// SIMATIC S7-200 SMART project (STEP 7-Micro/WIN SMART), CPU SR40

SYMBOL_TABLE 表格 1
流速               VD116
管道内静压            VD112
管道内温度            VD108
管道内部压差值          VD104
粉尘浓度值            VD100
END_SYMBOL_TABLE

SYMBOL_TABLE 系统符号
Always_On        SM0.0    // 始终接通
END_SYMBOL_TABLE

ORGANIZATION_BLOCK MAIN:OB1
TITLE=程序注释
BEGIN
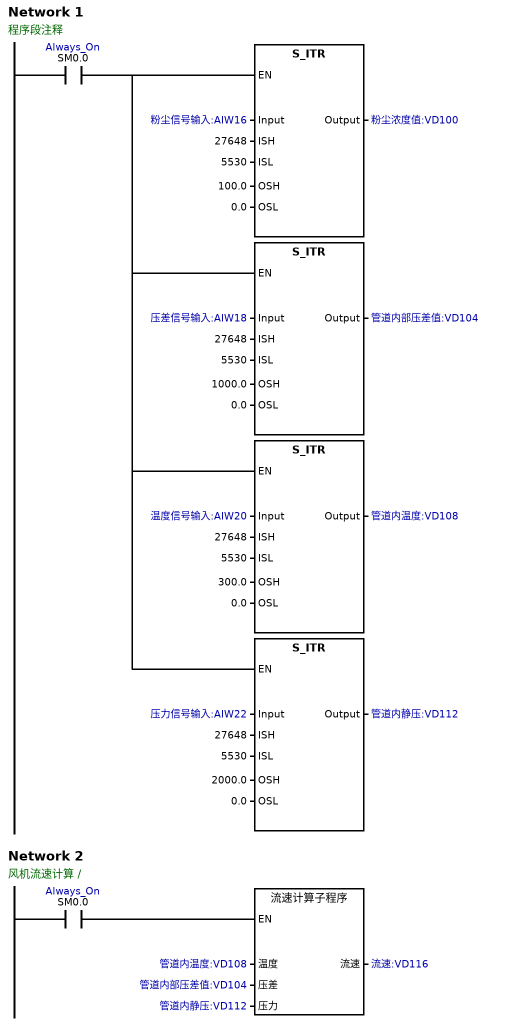
Network 1
// 程序段注释
LD     Always_On:SM0.0
CALL   S_ITR:SBR1, 粉尘信号输入:AIW16, 27648, 5530, 100.0, 0.0, 粉尘浓度值:VD100
CALL   S_ITR:SBR1, 压差信号输入:AIW18, 27648, 5530, 1000.0, 0.0, 管道内部压差值:VD104
CALL   S_ITR:SBR1, 温度信号输入:AIW20, 27648, 5530, 300.0, 0.0, 管道内温度:VD108
CALL   S_ITR:SBR1, 压力信号输入:AIW22, 27648, 5530, 2000.0, 0.0, 管道内静压:VD112
Network 2
// 风机流速计算
// 
LD     Always_On:SM0.0
CALL   流速计算子程序:SBR0, 管道内温度:VD108, 管道内部压差值:VD104, 管道内静压:VD112, 流速:VD116
END_ORGANIZATION_BLOCK

SUBROUTINE_BLOCK 流速计算子程序:SBR0
TITLE=子程序注释
VAR_INPUT
温度:REAL;	// LD0 
压差:REAL;	// LD4 
压力:REAL;	// LD8 
END_VAR
VAR_OUTPUT
流速:REAL;	// LD12 
END_VAR
VAR
Temp1:REAL;	// LD16 
END_VAR
BEGIN
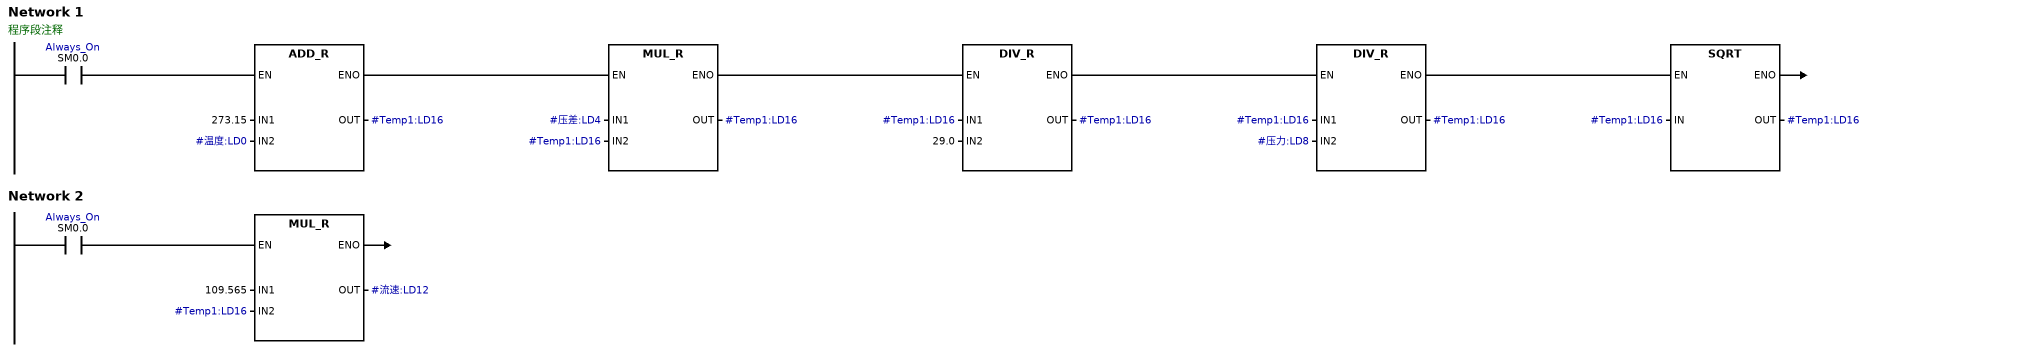
Network 1
// 程序段注释
LD     Always_On:SM0.0
MOVR   273.15, #Temp1:LD16
AENO
+R     #温度:LD0, #Temp1:LD16
AENO
*R     #压差:LD4, #Temp1:LD16
AENO
/R     29.0, #Temp1:LD16
AENO
/R     #压力:LD8, #Temp1:LD16
AENO
SQRT   #Temp1:LD16, #Temp1:LD16
Network 2
LD     Always_On:SM0.0
MOVR   109.565, #流速:LD12
*R     #Temp1:LD16, #流速:LD12
END_SUBROUTINE_BLOCK

// SBR1: protected block, not included
